# EPICS substitutions: streakcameraApp/Db/c5680.substitutions
file gen_params.template {
    {}
}

file img_params.template {
    {}
}

file ioc_control.template {
    {}
}

file operation.template {
    {}
}
